      BUFFER_4:
        IF (_nQueue[BUFFER_1] < 12)
        THEN
          _eState                             := E_PROGRESS.PROGRESS_PREPARE;
        END_IF
    END_CASE
END_CASE
//-----------------------------------------------------------------------------
//-----------------------------------------------------------------------------
CASE _eState
OF
  E_PROGRESS.PROGRESS_PREPARE:
    CASE _nProcess
    OF
      BUFFER_1:
        _bSparse                              := FALSE;
        IF (_nQueue[INPUT] = 0)
        THEN
          _nInputLastTarget                   := 0;
          _ItfProcess[BUFFER_1].TargetMask    := _wProcessInputMask;
          _eState                             := E_PROGRESS.PROGRESS_WORKING;
        END_IF
    ELSE
      _eState                                 := E_PROGRESS.PROGRESS_WORKING;
    END_CASE

END_CASE
//-----------------------------------------------------------------------------
//-----------------------------------------------------------------------------
CASE _eState
OF
  E_PROGRESS.PROGRESS_WORKING:

  CASE _eProcessState
  OF
    E_STATION_STATE.STATION_INIT:
      CASE _nProcess
      OF
        BUFFER_3:
          IF (_nQueue[OUTPUT_R1] = QUEUE_COUNT)
          THEN
            _eState                           := E_PROGRESS.PROGRESS_INIT;
          ELSE
            _eProcessCmd                      := E_STATION_CTRL.STATION_DISABLE;
          END_IF
      ELSE
        _eProcessCmd                          := E_STATION_CTRL.STATION_DISABLE;
      END_CASE

    E_STATION_STATE.STATION_DISABLE:
      _eProcessCmd                            := E_STATION_CTRL.STATION_ENABLE;

    E_STATION_STATE.STATION_MOVER_ENTER:
      CASE _ItfProcess[_nProcess].ProcessType
      OF
        E_PROCESS_TYPE.DISTRIBUTOR:
          CASE _nProcess
          OF
            BUFFER_4,
            DISTRIBUTOR_2,
            DISTRIBUTOR_1:
            IF (GVL_XTS.StationState[_ItfProcess[_nProcess].StationFirst].rMoverModPos > GVL_XTS.StationParameter[_ItfProcess[_nProcess].StationFirst].rPosWait-5.0)
            THEN
              _eState                           := E_PROGRESS.PROGRESS_OCCUPIED;
              _eProcessCmd                      := E_STATION_CTRL.STATION_MOVER_SEND;
            END_IF
          ELSE
            _eState                           := E_PROGRESS.PROGRESS_OCCUPIED;
            _eProcessCmd                      := E_STATION_CTRL.STATION_MOVER_SEND;
          END_CASE
(*
          IF (GVL_XTS.StationState[_ItfProcess[_nProcess].StationFirst].rMoverModPos > GVL_XTS.StationParameter[_ItfProcess[_nProcess].StationFirst].rPosWait-5.0)
          THEN
            _eState                           := E_PROGRESS.PROGRESS_OCCUPIED;
            _eProcessCmd                      := E_STATION_CTRL.STATION_MOVER_SEND;
          END_IF
*)
      ELSE
          _eProcessCmd                        := E_STATION_CTRL.STATION_MOVER_ENTER;
      END_CASE

    E_STATION_STATE.STATION_PROCESS_START:
      _tonProcess(IN := FALSE, PT := _tProcess);
      CASE _nProcess
      OF
        INPUT:
          IF (_nQueue[INPUT] = QUEUE_COUNT)
          THEN
            _eProcessCmd                      := E_STATION_CTRL.STATION_PROCESS_START;
          END_IF

        OUTPUT_R1,
        OUTPUT_R2:
          IF (_ItfProcess[OUTPUT_R1].ProcessState = _ItfProcess[OUTPUT_R2].ProcessState)
          THEN
            _eProcessCmd                      := E_STATION_CTRL.STATION_PROCESS_START;
          END_IF
      ELSE
        _eProcessCmd                          := E_STATION_CTRL.STATION_PROCESS_START;
      END_CASE


    E_STATION_STATE.STATION_PROCESS_DONE:
      _tonProcess(IN := TRUE, PT := _tProcess);

      IF _tonProcess.Q
      THEN
        _eProcessCmd                          := E_STATION_CTRL.STATION_PROCESS_DONE;
      END_IF

    E_STATION_STATE.STATION_MOVER_OUT:
      CASE _nProcess
      OF
        BUFFER_1:
          _eState                             := E_PROGRESS.PROGRESS_CHECK;

        Buffer_4:
          _eProcessCmd                        := E_STATION_CTRL.STATION_MOVER_OUT;
          IF (_nQueue[BUFFER_1] = QUEUE_COUNT-1)
          THEN
            _eState                           := E_PROGRESS.PROGRESS_INIT;
          END_IF

        BUFFER_3: 
          _eProcessCmd                        := E_STATION_CTRL.STATION_MOVER_OUT;


        OUTPUT_R1,
        OUTPUT_R2:
          IF (_ItfProcess[OUTPUT_R1].ProcessState = E_STATION_STATE.STATION_MOVER_OUT) AND
             (_ItfProcess[OUTPUT_R2].ProcessState = E_STATION_STATE.STATION_MOVER_OUT)
          THEN
            _eState                           := E_PROGRESS.PROGRESS_INIT;
            _eProcessCmd                      := E_STATION_CTRL.STATION_MOVER_OUT;
          END_IF

      ELSE
          _eState                             := E_PROGRESS.PROGRESS_INIT;
          _eProcessCmd                        := E_STATION_CTRL.STATION_MOVER_OUT;
      END_CASE
  END_CASE

END_CASE
//-----------------------------------------------------------------------------
//-----------------------------------------------------------------------------
CASE _eState
OF
  E_PROGRESS.PROGRESS_OCCUPIED:
      CASE _nProcess
      OF
        BUFFER_1:
          CASE _eProcessState
          OF
            E_STATION_STATE.STATION_MOVER_OUT:
            _wBufferSentMask                  := _ItfProcess[_nProcess].SetBitDWord(_wBufferSentMask, _nInputLastTarget);
            _nInputLastTarget                 := _nInputLastTarget + 1;
            _eState                           := E_PROGRESS.PROGRESS_WORKING;
          END_CASE
      ELSE
        _eState                               := E_PROGRESS.PROGRESS_WORKING;
      END_CASE
END_CASE
//-----------------------------------------------------------------------------
//-----------------------------------------------------------------------------
CASE _eState
OF
  E_PROGRESS.PROGRESS_CHECK:
    CASE _nProcess
    OF
      BUFFER_1:
        _eProcessCmd                          := E_STATION_CTRL.STATION_MOVER_OUT;
        IF (_wBufferSentMask = _wProcessInputMask)
        THEN
          _eState                             := E_PROGRESS.PROGRESS_INIT;
        ELSE
          _eState                             := E_PROGRESS.PROGRESS_WORKING;
        END_IF
    ELSE
      _eState                                 := E_PROGRESS.PROGRESS_INIT;
    END_CASE
END_CASE
//-----------------------------------------------------------------------------
//-----------------------------------------------------------------------------
_ItfProcess[_nProcess].ProcessCmd             := _eProcessCmd; 
AUTO                                          := _eState;
//-----------------------------------------------------------------------------
//-----------------------------------------------------------------------------
END_METHOD

METHOD AUTO_1 : E_PROGRESS
VAR_INPUT
  Active            : BOOL;
END_VAR
VAR_INST
  _bSparse            : Bool;
  _ncount             : uint;
  _eState,
  _eResult            : E_PROGRESS;

  _ndx                : UINT;

  _eProcessState      : E_STATION_STATE;
  _eProcessCmd        : E_STATION_CTRL;

  _nkx                : UINT;

  _nInputLastTarget   : UINT;

{attribute 'displaymode':='bin'}
  _wBufferSentMask    : dword;
{attribute 'displaymode':='bin'}
  _wProcessInputMask  : DWORD; // placement information for movers in stations from preceeding machine

  _eProcessType       : E_PROCESS_TYPE;
END_VAR
IF NOT Check() THEN AUTO_1 := E_PROGRESS.PROGRESS_ERROR; RETURN; END_IF

//-----------------------------------------------------------------------------
IF NOT Active 
THEN 
	_eState                                     := E_PROGRESS.PROGRESS_INIT;

  _nCount                                     := 0;
  memset(ADR(_nQueue), 0, SIZEOF(_nQueue));
  memset(ADR(_wProcessInputMask), 0, SIZEOF(_wProcessInputMask));
  memset(ADR(_wBufferSentMask), 0, SIZEOF(_wBufferSentMask));
ELSE
  _eProcessState                              := _ItfProcess[_nProcess].ProcessState;
  _eProcessType                               := _ItfProcess[_nProcess].ProcessType;

  FOR _ndx := 1 TO MAX_PROCESS
  DO
    _nQueue[_ndx]                             := _ItfProcess[_ndx].MoverCountInQueue;
  END_FOR
END_IF 
//-----------------------------------------------------------------------------
//-----------------------------------------------------------------------------
//-----------------------------------------------------------------------------
CASE _eState
OF
  E_PROGRESS.PROGRESS_INIT:
    IF Active
    THEN
      _nCount := _ncount + 1;
      _wProcessInputMask                      := 0;
      _wBufferSentMask                        := 0;
      _eState                                 := E_PROGRESS.PROGRESS_BUSY;
    END_IF
END_CASE
//-----------------------------------------------------------------------------
//-----------------------------------------------------------------------------
CASE _eState
OF
  E_PROGRESS.PROGRESS_BUSY:

    CASE _nProcess
    OF
      DISTRIBUTOR_2,
      DISTRIBUTOR_1:
        _eState                               := E_PROGRESS.PROGRESS_PREPARE;

      OUTPUT_R2:
        _eState                               := E_PROGRESS.PROGRESS_PREPARE;

      OUTPUT_R1:
        _eState                               := E_PROGRESS.PROGRESS_PREPARE;

      BUFFER_3:
        IF (_nQueue[_nProcess] > 11)
        THEN
          _eState                             := E_PROGRESS.PROGRESS_PREPARE;
        END_IF

      OUTPUT_1:
        _eState                               := E_PROGRESS.PROGRESS_PREPARE;

      INPUT:
        _eState                               := E_PROGRESS.PROGRESS_PREPARE;

      BUFFER_1:
        _eState                               := E_PROGRESS.PROGRESS_PREPARE;
        IF NOT _bSparse
        THEN
          FOR _nkx := 1 TO _ItfProcess[INPUT].StationCount
          DO
              _wProcessInputMask              := _ItfProcess[BUFFER_1].SetBitDWord(_wProcessInputMask, _nkx-1);
          END_FOR
        ELSE
          FOR _nkx := 1 TO _ItfProcess[INPUT].StationCount
          DO
            IF (_nkx <> 7)
            THEN
              _wProcessInputMask              := _ItfProcess[BUFFER_1].SetBitDWord(_wProcessInputMask, _nkx-1);
            END_IF
          END_FOR

        END_IF


      BUFFER_4:
        IF (_nQueue[BUFFER_1] < 8)
        THEN
          _eState                             := E_PROGRESS.PROGRESS_PREPARE;
        END_IF
    END_CASE
END_CASE
//-----------------------------------------------------------------------------
//-----------------------------------------------------------------------------
CASE _eState
OF
  E_PROGRESS.PROGRESS_PREPARE:
    CASE _nProcess
    OF
      BUFFER_1:
        _bSparse                              := FALSE;
        IF (_nQueue[INPUT] = 0)
        THEN
          _nInputLastTarget                   := 0;
          _ItfProcess[BUFFER_1].TargetMask    := _wProcessInputMask;
          _eState                             := E_PROGRESS.PROGRESS_WORKING;
        END_IF
    ELSE
      _eState                                 := E_PROGRESS.PROGRESS_WORKING;
    END_CASE

END_CASE
//-----------------------------------------------------------------------------
//-----------------------------------------------------------------------------
CASE _eState
OF
  E_PROGRESS.PROGRESS_WORKING:

  CASE _eProcessState
  OF
    E_STATION_STATE.STATION_INIT:
      _eProcessCmd                            := E_STATION_CTRL.STATION_DISABLE;

    E_STATION_STATE.STATION_DISABLE:
      _eProcessCmd                            := E_STATION_CTRL.STATION_ENABLE;

    E_STATION_STATE.STATION_MOVER_ENTER:
      CASE _eProcessType
      OF
        E_PROCESS_TYPE.DISTRIBUTOR:
          IF (GVL_XTS.StationState[_ItfProcess[_nProcess].StationFirst].rMoverModPos > GVL_XTS.StationParameter[_ItfProcess[_nProcess].StationFirst].rPosWait - 250.0)
          THEN
            _eState                           := E_PROGRESS.PROGRESS_OCCUPIED;
            _eProcessCmd                      := E_STATION_CTRL.STATION_MOVER_SEND;
          END_IF
      ELSE
          _eProcessCmd                        := E_STATION_CTRL.STATION_MOVER_ENTER;
      END_CASE

    E_STATION_STATE.STATION_PROCESS_START:
      _tonProcess(IN := FALSE, PT := _tProcess);
      _eProcessCmd                            := E_STATION_CTRL.STATION_PROCESS_START;


    E_STATION_STATE.STATION_PROCESS_DONE:
      _tonProcess(IN := TRUE, PT := _tProcess);

      IF _tonProcess.Q
      THEN
        _eProcessCmd                          := E_STATION_CTRL.STATION_PROCESS_DONE;
      END_IF

    E_STATION_STATE.STATION_MOVER_OUT:
      CASE _nProcess
      OF
        BUFFER_1:
          _eState                             := E_PROGRESS.PROGRESS_CHECK;

        Buffer_4:
          _eProcessCmd                        := E_STATION_CTRL.STATION_MOVER_OUT;
          IF (_nQueue[BUFFER_1] = QUEUE_COUNT-1)
          THEN
            _eState                           := E_PROGRESS.PROGRESS_INIT;
          END_IF

        BUFFER_3: 
          _eProcessCmd                        := E_STATION_CTRL.STATION_MOVER_OUT;
          IF (_nQueue[OUTPUT_R1] = QUEUE_COUNT)
          THEN
            _eState                           := E_PROGRESS.PROGRESS_INIT;
          END_IF


      ELSE
          _eState                             := E_PROGRESS.PROGRESS_INIT;
          _eProcessCmd                        := E_STATION_CTRL.STATION_MOVER_OUT;
      END_CASE
  END_CASE

END_CASE
//-----------------------------------------------------------------------------
//-----------------------------------------------------------------------------
CASE _eState
OF
  E_PROGRESS.PROGRESS_OCCUPIED:
      CASE _nProcess
      OF
        BUFFER_1:
          CASE _eProcessState
          OF
            E_STATION_STATE.STATION_MOVER_OUT:
            _wBufferSentMask                  := _ItfProcess[_nProcess].SetBitDWord(_wBufferSentMask, _nInputLastTarget);
            _nInputLastTarget                 := _nInputLastTarget + 1;
            _eState                           := E_PROGRESS.PROGRESS_WORKING;
          END_CASE
      ELSE
        _eState                               := E_PROGRESS.PROGRESS_WORKING;
      END_CASE
END_CASE
//-----------------------------------------------------------------------------
//-----------------------------------------------------------------------------
CASE _eState
OF
  E_PROGRESS.PROGRESS_CHECK:
    CASE _nProcess
    OF
      BUFFER_1:
        _eProcessCmd                          := E_STATION_CTRL.STATION_MOVER_OUT;
        IF (_wBufferSentMask = _wProcessInputMask)
        THEN
          _ItfProcess[BUFFER_1].TargetMask    := 0;
          _eState                             := E_PROGRESS.PROGRESS_INIT;
        ELSE
          _eState                             := E_PROGRESS.PROGRESS_WORKING;
        END_IF
    ELSE
      _eState                                 := E_PROGRESS.PROGRESS_INIT;
    END_CASE
END_CASE
//-----------------------------------------------------------------------------
//-----------------------------------------------------------------------------
_ItfProcess[_nProcess].ProcessCmd             := _eProcessCmd; 
AUTO_1                                          := _eState;
//-----------------------------------------------------------------------------
//-----------------------------------------------------------------------------
END_METHOD

METHOD Check : BOOL
VAR_INST
  _sCheck   : STRING;
  _nIdx     : UINT;
END_VAR

FOR _nIdx := 1 TO MAX_PROCESS
DO
  IF NOT (_ItfProcess[_nIdx] <> 0)
  THEN
    _sCheck   := concat('Invalid Interface Pointer at Index: ', TO_STRING(_nIdx));
    RETURN;
  END_IF
END_FOR

IF NOT (_nProcess > 0)
THEN
  _sCheck         := concat('NULL Invalid Index: ', TO_STRING(_nProcess));
  RETURN;
END_IF

IF (_nProcess > MAX_PROCESS)
THEN
  _sCheck         := concat('MAX Invalid Index: ', TO_STRING(_nProcess));
  RETURN;
END_IF

_nMoverPerMinute  := _ItfProcess[_nProcess].ProcessPerMinute;
_wTargetMask      := _ItfProcess[_nProcess].TargetMask;

Check             := TRUE;
END_METHOD

PROPERTY ItfProcesses : reference to ARRAY[1..MAX_PROCESS] OF I_ExternControl_Process
SET
_ItfProcess REF= ItfProcesses;
END_SET
END_PROPERTY

PROPERTY ProcessIndex : uint
GET
ProcessIndex  := _nProcess;
END_GET
SET
_nProcess   := ProcessIndex;
END_SET
END_PROPERTY

PROPERTY ProcessTime : time
GET
ProcessTime := _tProcess;
END_GET
SET
_tProcess := ProcessTime;
END_SET
END_PROPERTY

METHOD RESET : E_PROGRESS
VAR_INPUT
  Execute         : BOOL;
END_VAR
VAR
  _eState,
  _eResult          : E_PROGRESS;
END_VAR

//-----------------------------------------------------------------------------
IF NOT Execute 
THEN 
	_eState                                     := E_PROGRESS.PROGRESS_INIT; 
END_IF 
//-----------------------------------------------------------------------------
//-----------------------------------------------------------------------------
//-----------------------------------------------------------------------------
CASE _eState
OF
  E_PROGRESS.PROGRESS_INIT:
    IF Execute
    THEN
      IF NOT (_ItfProcess[_nProcess] <> 0)
      THEN
        _eState                               := E_PROGRESS.PROGRESS_ERROR;
      ELSE
        _eState                               := E_PROGRESS.PROGRESS_BUSY;
      END_IF
    END_IF
END_CASE
//-----------------------------------------------------------------------------
//-----------------------------------------------------------------------------
CASE _eState
OF
  E_PROGRESS.PROGRESS_BUSY:
    _eState                                   := E_PROGRESS.PROGRESS_PREPARE;
END_CASE
//-----------------------------------------------------------------------------
//-----------------------------------------------------------------------------
CASE _eState
OF
  E_PROGRESS.PROGRESS_PREPARE:
    IF (_ItfProcess[_nProcess].Init())
    THEN
      _eState                                 := E_PROGRESS.PROGRESS_DONE;
    END_IF
END_CASE
//-----------------------------------------------------------------------------
//-----------------------------------------------------------------------------
END_METHOD

END_FUNCTION_BLOCK

// ---- GlobalTextList.TcGTLO
TEXTLIST GlobalTextList
  448 = ' %s'
  360 = ' Application Processes:'
  17 = ' STATION_ENABLE'
  34 = ' STATION_MOVER_ENTER'
  452 = ' STATION_MOVER_GONE'
  75 = ' STATION_MOVER_OUT'
  598 = ' STATION_PROCESS_DONE'
  750 = ' STATION_PROCESS_START'
  632 = ' XTS Stations:'
  294 = '%.2f'
  191 = '%d'
  836 = '%s'
  704 = 'All Positions Valid'
  562 = 'AllAxisStanding'
  784 = 'Application/Process'
  878 = 'AxisCount Enabled: %d'
  162 = 'AxisCount: %d'
  951 = 'Command'
  914 = 'ConstantVelocity'
  929 = 'Control'
  707 = 'CyclicCheck: %s'
  660 = 'DC Link All Modules'
  359 = 'Decelerating'
  843 = 'Detected AxisCount: %d'
  698 = 'Enabled'
  918 = 'EnableProcess'
  510 = 'eState'
  772 = 'Expected AxisCount: %d'
  48 = 'GroupDisabled'
  915 = 'GroupError'
  495 = 'GroupErrorId: %d'
  975 = 'GroupErrorStop'
  940 = 'GroupHoming'
  300 = 'GroupMoving'
  807 = 'GroupNotReady'
  438 = 'GroupStandby'
  226 = 'GroupStatusBusy'
  204 = 'GroupStatusValid'
  973 = 'GroupStopping'
  505 = 'GVL_XTS.'
  942 = 'GVL_XTS.CaGroupInfo'
  611 = 'GVL_XTS.XtsTransportState.GroupInfo'
  680 = 'ID Detection Active'
  238 = 'ID Detection Error'
  526 = 'ID Detection Mode: %s'
  29 = 'ID Detection Valid'
  211 = 'Info Act Pos Absolute'
  586 = 'Info Act Pos Modulo'
  21 = 'Info Mover Avoiding Collision'
  282 = 'Info Mover Coupled'
  398 = 'Info Mover Enabled'
  751 = 'Info Mover Error'
  907 = 'Info Mover Standstill'
  480 = 'Info nError ID'
  922 = 'Info Target Pos Absolute'
  16 = 'Info Target Pos Modulo'
  616 = 'InPosition'
  779 = 'Mask: %s'
  726 = 'McGroupState:      %s'
  974 = 'MOVER command'
  387 = 'Mover ID: %d'
  297 = 'Mover Position Assignement: %s'
  840 = 'MOVER result:  %s'
  53 = 'MOVER state:   %s'
  502 = 'nMask'
  232 = 'nMoverId'
  756 = 'nMoverSelected: %d'
  371 = 'nQueue'
  427 = 'Offset: %.3f'
  312 = 'Operation Mode: %s'
  143 = 'Process'
  423 = 'ProcessCmd'
  861 = 'ProcessState'
  320 = 'Queue: %d'
  91 = 'Set Acceleration'
  399 = 'Set Delta'
  382 = 'Set Distance'
  757 = 'Set Gap'
  934 = 'Set Jerk'
  201 = 'Set Override'
  936 = 'Set Position'
  62 = 'Set Velocity'
  231 = 'State'
  567 = 'Target Station: %d'
  993 = 'Type'
  275 = 'XPU Command'
  227 = 'XpuResult:   %s'
  96 = 'XpuState:    %s'
  884 = 'XTS Station'
  377 = 'XTS Stations Enabled'
  572 = 'XTS Transport Check:  %s'
  500 = 'XTS Transport Command'
  395 = 'XTS Transport Result: %s'
  798 = 'XTS Transport State:  %s'
  568 = 'XTS_Transport. GroupInfo'
  413 = 'XTS_Transport.GroupInfo'
END_TEXTLIST

// ---- PROCESS/_Visualization/T_PROCESS_VISU.TcVIS
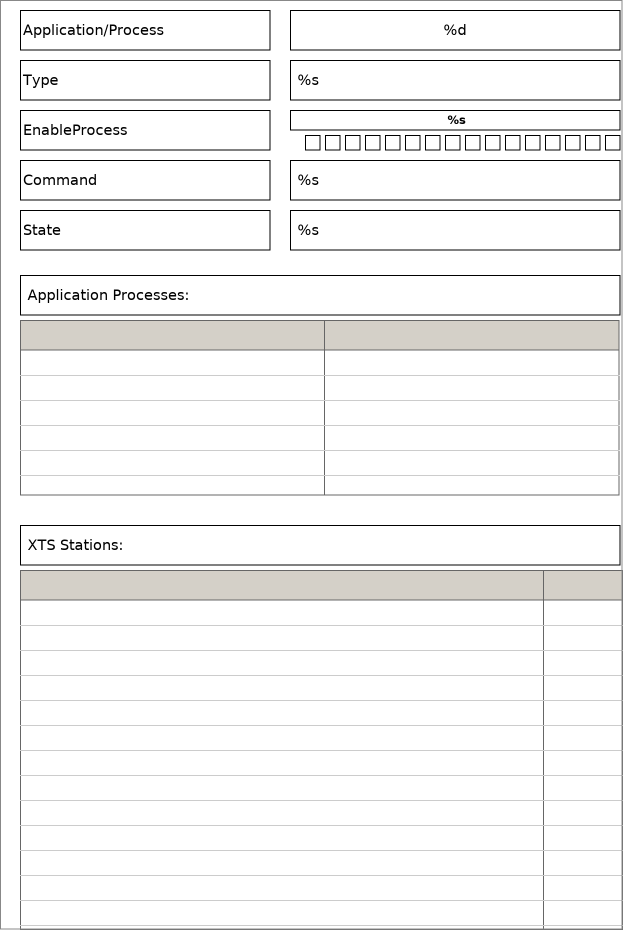
VISUALIZATION T_PROCESS_VISU  // 623x930
VAR_IN_OUT
	nSelectedProcess    : UINT; // selected process index
  EnableProcess       : ARRAY[1..GVL_PROCESS.MAX_PROCESS] OF WORD;
  ProcessCmd          : ARRAY[1..GVL_PROCESS.MAX_PROCESS] OF E_STATION_CTRL;
  ProcessState        : ARRAY[1..GVL_PROCESS.MAX_PROCESS] OF E_STATION_STATE;
  StationState        : ARRAY[1..MAX_STATION] OF ST_STATION_STATE;
  bStationEnabled     : ARRAY[1..MAX_STATION] OF BOOL;
END_VAR
    Rectangle (20,10 250x40), "Application/Process"
    Rectangle (290,10 330x40), "%d", text variable: nSelectedProcess
        OnMouseClick: write the text variable via VisuDialogs.Numpad, min 1, max GVL_PROCESS.MAX_PROCESS, title 'Selected Process'
    Rectangle (20,160 250x40), "Command"
    Rectangle (20,210 250x40), "State"
    Rectangle (20,60 250x40), "Type"
    Rectangle (20,110 250x40), "EnableProcess"
    Rectangle (290,60 330x40), "%s", text variable: GVL_PROCESS.Process[nSelectedProcess]._eType
    Rectangle (290,160 330x40), "%s", text variable: GVL_PROCESS.Process[nSelectedProcess]._eProcessCmd
    Rectangle (290,210 330x40), "%s", text variable: GVL_PROCESS.Process[nSelectedProcess]._eProcessState
    Rectangle (290,110 330x20), "%s", text variable: MAIN.sProcessEnableMask
    Rectangle (605,135 15x15)
        toggle EnableProcess[nSelectedProcess].0
    Rectangle (585,135 15x15)
        toggle EnableProcess[nSelectedProcess].1
    Rectangle (565,135 15x15)
        toggle EnableProcess[nSelectedProcess].2
    Rectangle (545,135 15x15)
        toggle EnableProcess[nSelectedProcess].3
    Rectangle (525,135 15x15)
        toggle EnableProcess[nSelectedProcess].4
    Rectangle (505,135 15x15)
        toggle EnableProcess[nSelectedProcess].5
    Rectangle (485,135 15x15)
        toggle EnableProcess[nSelectedProcess].6
    Rectangle (465,135 15x15)
        toggle EnableProcess[nSelectedProcess].7
    Table (20,570 540x360), data array: StationState
        p3854506369: StationState[INDEX].eState
        p1892666644: StationState[INDEX].nMask
        p338671338: StationState[INDEX].nMoverId
        p2170511999: StationState[INDEX].nQueue
    Table (543,570 80x360), data array: bStationEnabled
        p3854506369: bStationEnabled[INDEX]
    Rectangle (445,135 15x15)
        toggle EnableProcess[nSelectedProcess].8
    Rectangle (425,135 15x15)
        toggle EnableProcess[nSelectedProcess].9
    Rectangle (405,135 15x15)
        toggle EnableProcess[nSelectedProcess].10
    Rectangle (385,135 15x15)
        toggle EnableProcess[nSelectedProcess].11
    Rectangle (365,135 15x15)
        toggle EnableProcess[nSelectedProcess].12
    Rectangle (345,135 15x15)
        toggle EnableProcess[nSelectedProcess].13
    Rectangle (325,135 15x15)
        toggle EnableProcess[nSelectedProcess].14
    Rectangle (305,135 15x15)
        toggle EnableProcess[nSelectedProcess].15
    Rectangle (20,525 600x40), "XTS Stations:"
    Rectangle (20,275 600x40), "Application Processes:"
    Table (20,320 329x175), data array: ProcessState
        p3854506369: ProcessState[INDEX]
    Table (324,320 295x175), data array: ProcessCmd
        p3854506369: ProcessCmd[INDEX]
END_VISUALIZATION

// ---- PROCESS/_Visualization/PROCESS_XTS_TRANSPORT.TcVIS
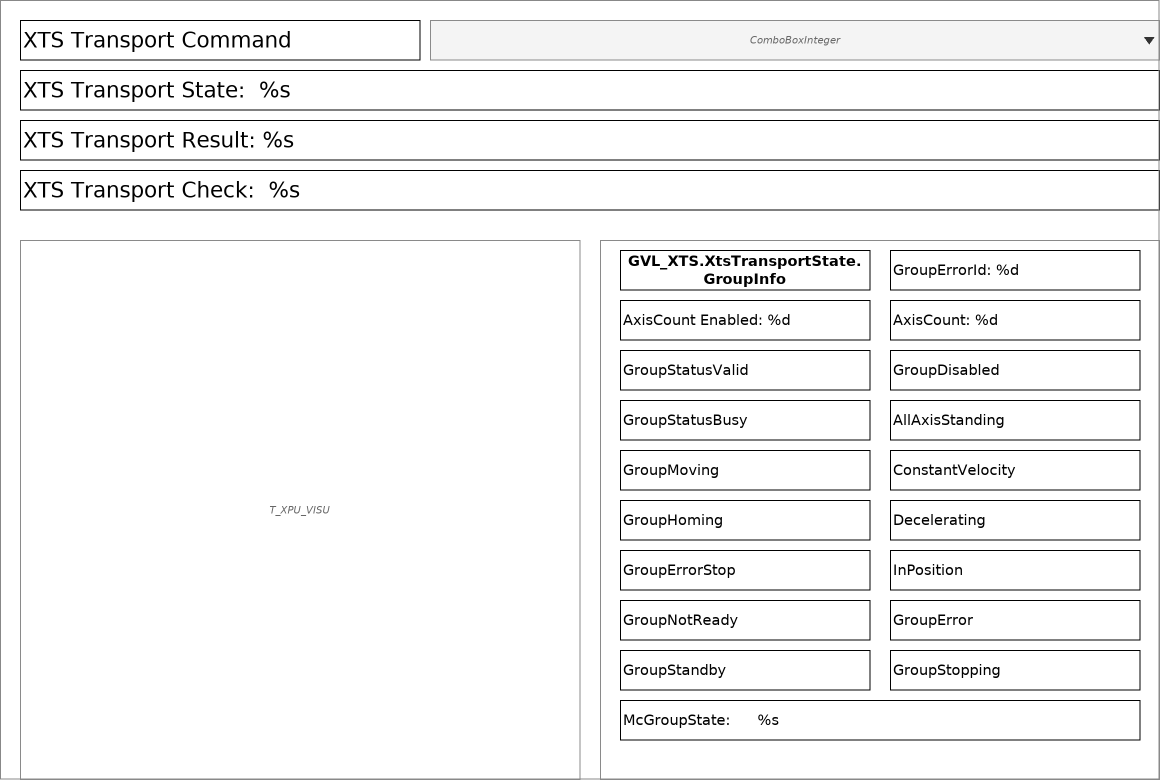
VISUALIZATION PROCESS_XTS_TRANSPORT  // 1160x780
    Rectangle (20,20 400x40), "XTS Transport Command"
    ComboBoxInteger (430,20 730x40), variable: GVL_XTS.XtsTransportCtrl.Cmd, text list: 'TL_E_CTRL_TRANSPORT'
    Frame (20,240 560x540)
        shows T_XPU_VISU()
    Frame (600,240 560x540)
        shows GROUP_VISU()
    Rectangle (20,70 1140x40), "XTS Transport State: %s", text variable: MAIN.sTransportState
    Rectangle (20,120 1140x40), "XTS Transport Result: %s", text variable: MAIN.sTransportResult
    Rectangle (20,170 1140x40), "XTS Transport Check: %s", text variable: MAIN.sTransportCheck
END_VISUALIZATION

// ---- XTS_TRANSPORT/_Visualization/GROUP_VISU.TcVIS
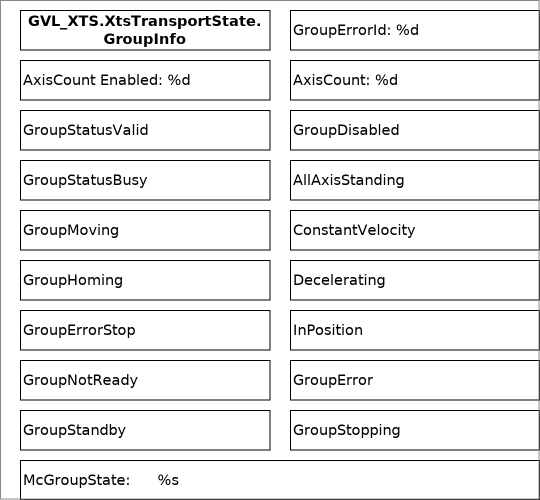
VISUALIZATION GROUP_VISU  // 540x500
    Rectangle (20,110 250x40), "GroupStatusValid", colour toggle: GVL_XTS.XtsTransportState.GroupInfo.GroupStatusValid
    Rectangle (20,160 250x40), "GroupStatusBusy", colour toggle: GVL_XTS.XtsTransportState.GroupInfo.GroupStatusBusy
    Rectangle (20,210 250x40), "GroupMoving", colour toggle: GVL_XTS.XtsTransportState.GroupInfo.GroupMoving
    Rectangle (20,260 250x40), "GroupHoming", colour toggle: GVL_XTS.XtsTransportState.GroupInfo.GroupHoming
    Rectangle (20,310 250x40), "GroupErrorStop", colour toggle: GVL_XTS.XtsTransportState.GroupInfo.GroupErrorStop
    Rectangle (20,360 250x40), "GroupNotReady", colour toggle: GVL_XTS.XtsTransportState.GroupInfo.GroupNotReady
    Rectangle (20,410 250x40), "GroupStandby", colour toggle: GVL_XTS.XtsTransportState.GroupInfo.GroupStandby
    Rectangle (290,410 250x40), "GroupStopping", colour toggle: GVL_XTS.XtsTransportState.GroupInfo.GroupStopping
    Rectangle (290,110 250x40), "GroupDisabled", colour toggle: GVL_XTS.XtsTransportState.GroupInfo.GroupDisabled
    Rectangle (290,160 250x40), "AllAxisStanding", colour toggle: GVL_XTS.XtsTransportState.GroupInfo.AllAxesStanding
    Rectangle (290,210 250x40), "ConstantVelocity", colour toggle: GVL_XTS.XtsTransportState.GroupInfo.ConstantVelocity
    Rectangle (290,260 250x40), "Decelerating", colour toggle: GVL_XTS.XtsTransportState.GroupInfo.Decelerating
    Rectangle (290,310 250x40), "InPosition", colour toggle: GVL_XTS.XtsTransportState.GroupInfo.InPosition
    Rectangle (290,360 250x40), "GroupError", colour toggle: GVL_XTS.XtsTransportState.GroupInfo.GroupError
    Rectangle (290,10 250x40), "GroupErrorId: %d", text variable: GVL_XTS.XtsTransportState.GroupInfo.GroupErrorId
    Rectangle (290,60 250x40), "AxisCount: %d", text variable: GVL_XTS.XtsTransportState.GroupInfo.AxisCount
    Rectangle (20,10 250x40), "GVL_XTS.XtsTransportState.GroupInfo"
    Rectangle (20,460 520x40), "McGroupState: %s", text variable: MAIN.sCaGroupState
    Rectangle (20,60 250x40), "AxisCount Enabled: %d", text variable: GVL_XTS.XtsTransportState.GroupInfo.AxisCountEnabled
END_VISUALIZATION

// ---- XTS_TRANSPORT/_Visualization/textlists/TL_E_CTRL_STATION.TcTLO
TEXTLIST TL_E_CTRL_STATION
  0 = 'STATION_CTRL_NULL'
  1 = 'STATION_INIT'
  10 = 'STATION_DISABLE'
  11 = 'STATION_ENABLE'
  20 = 'STATION_MOVER_ENTER'
  21 = 'STATION_MOVER_ENTER_RETRY'
  22 = 'STATION_MOVER_SEND'
  30 = 'STATION_PROCESS_START'
  31 = 'STATION_PROCESS_DONE'
  50 = 'STATION_MOVER_OUT'
  51 = 'STATION_MOVER_OUT_RETRY'
  60 = 'STATION_MOVER_GONE'
   = ''
END_TEXTLIST

// ---- XTS_TRANSPORT/_Visualization/textlists/TL_E_CTRL_XPU.TcTLO
TEXTLIST TL_E_CTRL_XPU
  0 = 'XTS_CMD_NULL'
  10 = 'XTS_CMD_INIT'
  30 = 'XTS_IDLE'
   = ''
END_TEXTLIST
